FUNCTION_BLOCK PUBLLP8 (* A proxy to 8-Variable local Publisher with interface of global publisher and logic outputs *)
  (* Standard: 61499-1; Classification: Communications *)
  (* Version 0.0, 2000-03-31, JHC, Rockwell Automation *)
  (* Compiler header: package fb.rt.vnet;import fb.rt.net.*; *)
  (* Compiler Java IBM VisualAge 3.0 *)
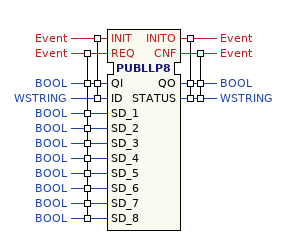
  EVENT_INPUT
    INIT WITH QI, ID; (* Service Initialization *)
    REQ WITH QI, SD_1, SD_2, SD_3, SD_4, SD_5, SD_6, SD_7, SD_8; (* Service Request *)
  END_EVENT
  EVENT_OUTPUT
    INITO WITH QO, STATUS; (* Initialization Confirm *)
    CNF WITH QO, STATUS; (* Service Confirmation *)
  END_EVENT
  VAR_INPUT
    QI : BOOL; (* Event Input Qualifier *)
    ID : WSTRING; (* Connection Identifier *)
    SD_1 : BOOL; (* Data to Send *)
    SD_2 : BOOL; (* Data to Send *)
    SD_3 : BOOL; (* Data to Send *)
    SD_4 : BOOL; (* Data to Send *)
    SD_5 : BOOL; (* Data to Send *)
    SD_6 : BOOL; (* Data to Send *)
    SD_7 : BOOL; (* Data to Send *)
    SD_8 : BOOL; (* Data to Send *)
  END_VAR
  VAR_OUTPUT
    QO : BOOL; (* Event Output Qualifier *)
    STATUS : WSTRING; (* Service Status *)
  END_VAR
  FBS
    PUBL : PUBL_8;
  END_FBS
  EVENT_CONNECTIONS
    INIT TO PUBL.INIT;
    REQ TO PUBL.REQ;
    PUBL.INITO TO INITO;
    PUBL.CNF TO CNF;
  END_CONNECTIONS
  DATA_CONNECTIONS
    ID TO PUBL.ID;
    SD_1 TO PUBL.SD_1;
    SD_2 TO PUBL.SD_2;
    SD_3 TO PUBL.SD_3;
    SD_4 TO PUBL.SD_4;
    SD_5 TO PUBL.SD_5;
    SD_6 TO PUBL.SD_6;
    SD_7 TO PUBL.SD_7;
    SD_8 TO PUBL.SD_8;
  END_CONNECTIONS
END_FUNCTION_BLOCK
